{attribute 'OPC.UA.DA.StructuredType' := '1'}
FUNCTION_BLOCK FB_Sensor_4_20mA_Generic EXTENDS FB_BaseDevice IMPLEMENTS I_Device, I_Sensor

VAR
	{attribute 'OPC.UA.DA' := '1'} 
	eSensorType: E_SensorType;
	{attribute 'OPC.UA.DA' := '0'} 
	nRawInput AT %I*: INT;
	{attribute 'OPC.UA.DA' := '1'} 
	nCurrentValue: REAL;
	
	{attribute 'OPC.UA.DA' := '1'} 
	nVal4mA: REAL;
	{attribute 'OPC.UA.DA' := '1'} 
	nVal20mA: REAL;
END_VAR

calculate();

METHOD calculate : BOOL
VAR_INPUT
END_VAR
nCurrentValue := nVal4mA + (INT_TO_REAL(nRawInput) / GVL.nMaxADCOutput) * (nVal20mA - nVal4mA) ;
END_METHOD

{warning 'add method implementation '}
METHOD disable : BOOL
bEnable := FALSE;
END_METHOD

{warning 'add method implementation '}
METHOD enable : BOOL
bEnable := TRUE;
END_METHOD

{warning 'add method implementation '}
METHOD FB_init : BOOL
VAR_INPUT
	(* if TRUE, the retain variables are initialized (warm start / cold start)*)
	bInitRetains	: BOOL;
	(* if TRUE, the instance afterwards gets moved into the copy code (online change)*)
	bInCopyCode	: BOOL;
	SensorID	: STRING(80);
	SensorDescr	: STRING(255);
	SensorType	: E_SensorType;
	

END_VAR
sID := SensorID;
sDescr := SensorDescr;
eSensorType := SensorType;
END_METHOD

{warning 'add method implementation '}
METHOD getType : E_SensorType
getType := eSensorType;
END_METHOD

{warning 'add method implementation '}
METHOD getValue : REAL
getValue := nCurrentValue;
END_METHOD

METHOD setLimits : BOOL
VAR_INPUT
	Val_4mA: 	REAL;
	Val_20mA: 	REAL;
END_VAR
nVal4mA := Val_4mA;
nVal20mA := Val_20mA;
END_METHOD

{warning 'add method implementation '}
METHOD write : BOOL
END_METHOD

END_FUNCTION_BLOCK

(* stored: Version 1.1.0.1, ProductVersion 3.1.4024.12
   POU FB_Sensor_4_20mA_Generic: Id {c0927399-3adb-47b4-bf92-aa20a2b989cb}, SpecialFunc None
   Method calculate: Id {23a37c0f-3f49-4065-9f31-c1ede2725044}
   Method disable: Id {7406af38-0d0c-45b5-885b-1800b14dc2d6}
   Method enable: Id {25771364-7f4e-4b8c-a440-aaea871004f4}
   Method FB_init: Id {e743491d-7c4d-4846-8a3e-febc368c23ce}
   Method getType: Id {374732ee-0a91-48e3-bc13-844523f9b29c}
   Method getValue: Id {a8673510-9521-469e-a4b3-2471be363ec9}
   Method setLimits: Id {7253a6e8-5688-4c6a-9e28-5c8d523cd39a}
   Method write: Id {0c7d7757-117b-44e1-a2db-fc685086cb20} *)
